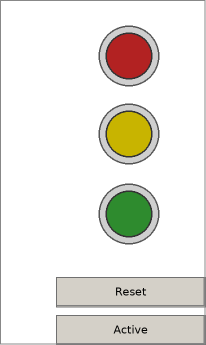
VISUALIZATION Ampel  // 206x345
    Lamp1 (94,21 70x70), variable: GVL_HMI_Ampel.LED_Rot, style: Lamp-Lamp1-Red
    Lamp1 (94,99 70x70), variable: GVL_HMI_Ampel.LED_Gelb, style: Lamp-Lamp1-Yellow
    Lamp1 (94,179 70x70), variable: GVL_HMI_Ampel.LED_Gruen, style: Lamp-Lamp1-Green
    Button (56,277 150x30), "Reset"
        tap GVL_HMI_Ampel.btnReset
    Button (56,315 150x30), "Active"
        tap GVL_HMI_Ampel.btnActive
END_VISUALIZATION

(* stored: Version 1.1.0.1, ProductVersion 3.1.4024.12
   Visu Ampel: Id {47e57637-d8a3-405f-bebf-f3fc73924987} *)
